FUNCTION_BLOCK GearSequenceStop EXTENDS GearSequence IMPLEMENTS ZCore.ISequence
VAR
  _step : ZCore.Step(GearStep.StopBegin, GearStep.StopEnd);
  _timerSim : ZAux.Timer;
END_VAR

IF OnStart(_step) THEN
  ; // init custom sequence variables here ...
END_IF

REPEAT
  LogStep();

  CASE _step.Index OF
    (* -------------------------------------------------------------------------------------------------------------------------------- *)
    GearStep.StopBegin:
    (* -------------------------------------------------------------------------------------------------------------------------------- *)
      IF _step.OnEntry()
      THEN
        _axis.PositionX.StopAsync(THIS^);
        _axis.RotationC.StopAsync(THIS^);
      END_IF
      
      Await2( _axis.PositionX, _axis.RotationC, nextStep:=GearStep.StopEnd);

    (* -------------------------------------------------------------------------------------------------------------------------------- *)
    GearStep.StopEnd:
    (* -------------------------------------------------------------------------------------------------------------------------------- *)    
      SetBusy(FALSE);
  
  ELSE
    Abort('sequence contains unhandled step');
  END_CASE
UNTIL _step.IsNotRepeatable() OR_ELSE NOT Busy END_REPEAT

END_FUNCTION_BLOCK

(* stored: Version 1.1.0.1
   POU GearSequenceStop: Id {97ab607c-34a5-41ed-813e-8396f91d99f1}, SpecialFunc None *)
